PROGRAM Stn5DosingPumpCtrl

VAR

END_VAR

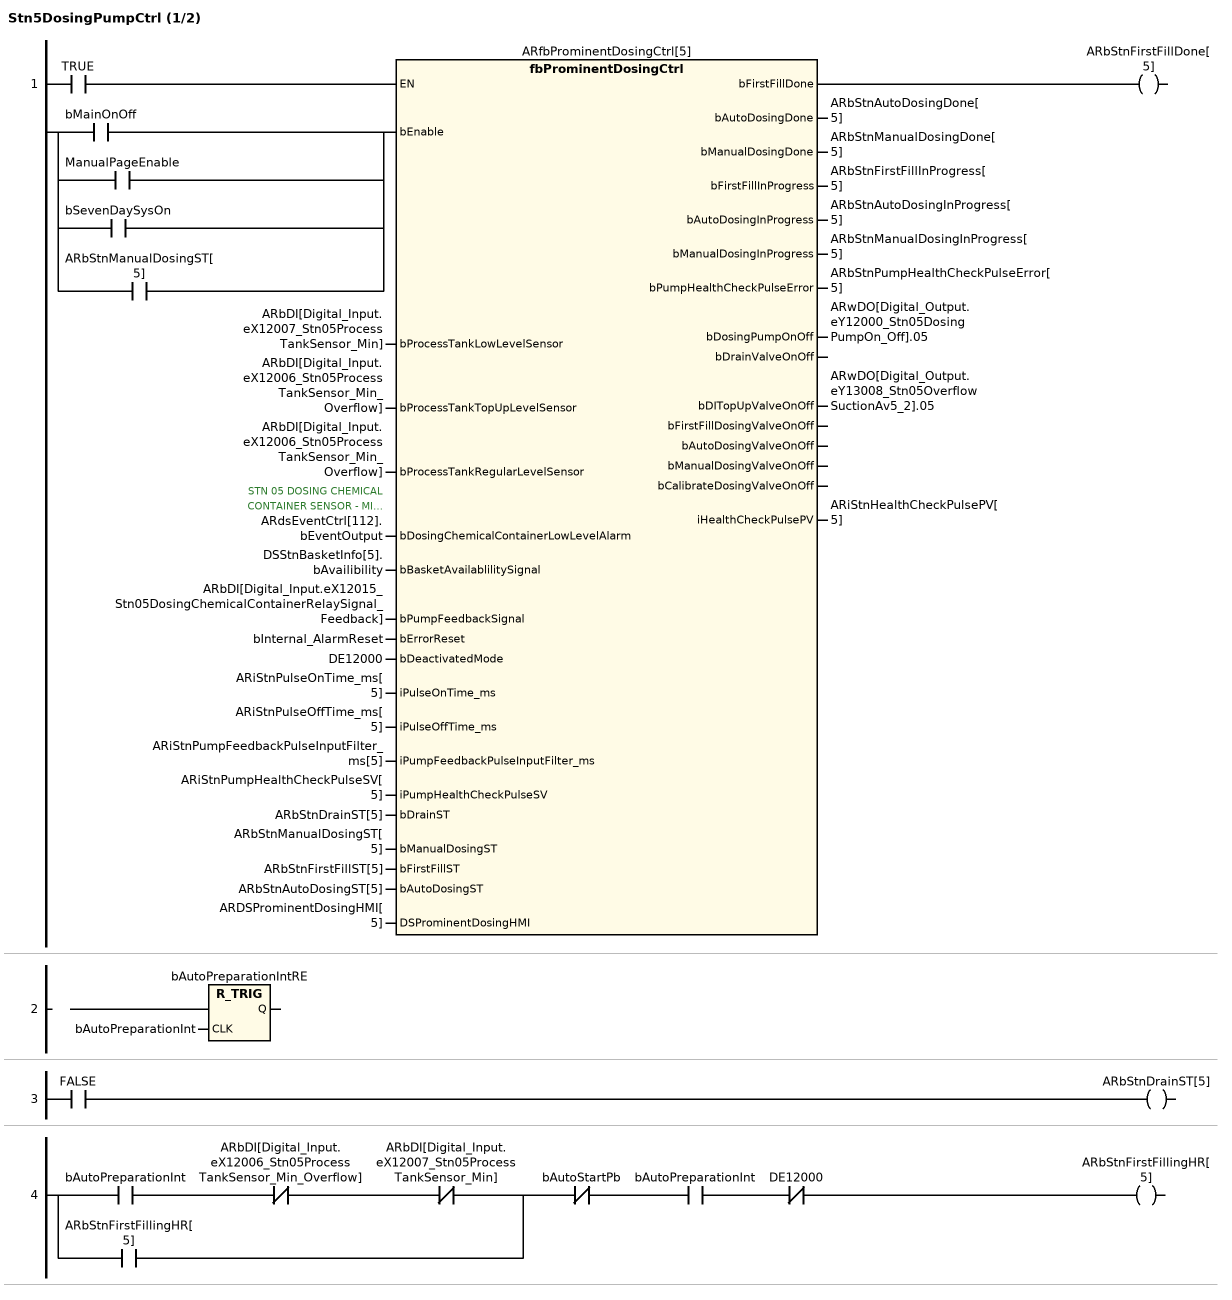
// NETWORK 1
//   ARdsEventCtrl[112].bEventOutput: STN 05 DOSING CHEMICAL CONTAINER SENSOR - MIN LEVEL
ARfbProminentDosingCtrl[5](
    bEnable := bMainOnOff OR ManualPageEnable OR bSevenDaySysOn OR ARbStnManualDosingST[5],
    bProcessTankLowLevelSensor := ARbDI[Digital_Input.eX12007_Stn05ProcessTankSensor_Min],
    bProcessTankTopUpLevelSensor := ARbDI[Digital_Input.eX12006_Stn05ProcessTankSensor_Min_Overflow],
    bProcessTankRegularLevelSensor := ARbDI[Digital_Input.eX12006_Stn05ProcessTankSensor_Min_Overflow],
    bDosingChemicalContainerLowLevelAlarm := ARdsEventCtrl[112].bEventOutput,
    bBasketAvailablilitySignal := DSStnBasketInfo[5].bAvailibility,
    bPumpFeedbackSignal := ARbDI[Digital_Input.eX12015_Stn05DosingChemicalContainerRelaySignal_Feedback],
    bErrorReset := bInternal_AlarmReset,
    bDeactivatedMode := DE12000,
    iPulseOnTime_ms := ARiStnPulseOnTime_ms[5],
    iPulseOffTime_ms := ARiStnPulseOffTime_ms[5],
    iPumpFeedbackPulseInputFilter_ms := ARiStnPumpFeedbackPulseInputFilter_ms[5],
    iPumpHealthCheckPulseSV := ARiStnPumpHealthCheckPulseSV[5],
    bDrainST := ARbStnDrainST[5],
    bManualDosingST := ARbStnManualDosingST[5],
    bFirstFillST := ARbStnFirstFillST[5],
    bAutoDosingST := ARbStnAutoDosingST[5],
    DSProminentDosingHMI := ARDSProminentDosingHMI[5],
    bAutoDosingDone => ARbStnAutoDosingDone[5],
    bManualDosingDone => ARbStnManualDosingDone[5],
    bFirstFillInProgress => ARbStnFirstFillInProgress[5],
    bAutoDosingInProgress => ARbStnAutoDosingInProgress[5],
    bManualDosingInProgress => ARbStnManualDosingInProgress[5],
    bPumpHealthCheckPulseError => ARbStnPumpHealthCheckPulseError[5],
    bDosingPumpOnOff => ARwDO[Digital_Output.eY12000_Stn05DosingPumpOn_Off].05,
    bDITopUpValveOnOff => ARwDO[Digital_Output.eY13008_Stn05OverflowSuctionAv5_2].05,
    iHealthCheckPulsePV => ARiStnHealthCheckPulsePV[5]); // fbProminentDosingCtrl
ARbStnFirstFillDone[5] := ARfbProminentDosingCtrl[5].bFirstFillDone;

// NETWORK 2
bAutoPreparationIntRE(CLK := bAutoPreparationInt); // R_TRIG

// NETWORK 3
ARbStnDrainST[5] := FALSE;

// NETWORK 4
ARbStnFirstFillingHR[5] := (bAutoPreparationInt AND NOT ARbDI[Digital_Input.eX12006_Stn05ProcessTankSensor_Min_Overflow] AND NOT ARbDI[Digital_Input.eX12007_Stn05ProcessTankSensor_Min] OR ARbStnFirstFillingHR[5]) AND NOT bAutoStartPb AND bAutoPreparationInt AND NOT DE12000;

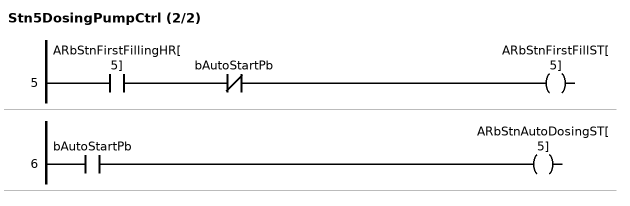
// NETWORK 5
ARbStnFirstFillST[5] := ARbStnFirstFillingHR[5] AND NOT bAutoStartPb;

// NETWORK 6
ARbStnAutoDosingST[5] := bAutoStartPb;

END_PROGRAM

(* stored: Version 1.1.0.1, ProductVersion 3.1.4024.12
   POU Stn5DosingPumpCtrl: Id {20bcb165-b392-444e-87fa-5380ace5649f}, SpecialFunc None *)
